{attribute 'pack_mode' := '2'}
TYPE ST_INSTANCE_CTRL :
STRUCT
  Cmd     : E_INSTANCE_CMD;
END_STRUCT
END_TYPE

(* stored: Version 1.1.0.1
   DUT ST_INSTANCE_CTRL: Id {cb04d147-9e4d-4a15-b8c5-35000f2ed7fa} *)
